RESOURCE_TYPE top
  (* Standard: 61499-2 *)
  (* Version 0.1, 2017-00-29, hpea485, UOA *)
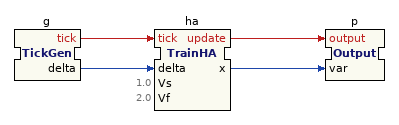
  FBS
    g : TickGen;
    ha : TrainHA(Vs := 1.0, Vf := 2.0);
    p : Output;
  END_FBS
  EVENT_CONNECTIONS
    g.tick TO ha.tick;
    ha.update TO p.output;
  END_CONNECTIONS
  DATA_CONNECTIONS
    g.delta TO ha.delta;
    ha.x TO p.var;
  END_CONNECTIONS
END_RESOURCE_TYPE
